// TIA Portal V20 export
DATA_BLOCK "IOLinkConfig"   // DB4000
{ S7_Optimized_Access := 'FALSE' }
// stored: AutoNumber false
   VAR
      "8B1.B" : "TypeIOLinkParamArray";   // sensor IO-Link adjustment scannerhousing
      "8B1" : "TypeIOLinkParamArray";   // sensor IO-Link light barrier measuring distance top
      "8B2" : "TypeIOLinkParamArray";   // sensor IO-Link light barrier measuring distance left
      "8B3" : "TypeIOLinkParamArray";   // sensor IO-Link light barrier measuring distance right
      Empty : "TypeIOLinkParamArray";
      "8B1.B-Restart-Conf" : Bool;   // sensor IO-Link adjustment scannerhousing - restart config
      "8B1-Restart-Conf" : Bool;   // sensor IO-Link light barrier measuring distance top - restart config
      "8B2-Restart-Conf" : Bool;   // sensor IO-Link light barrier measuring distance left - restart config
      "8B3-Restart-Conf" : Bool;   // sensor IO-Link light barrier measuring distance right - restart config
   END_VAR
BEGIN
END_DATA_BLOCK
